// TIA Portal V20 export
DATA_BLOCK "Interface"   // DB238
{ S7_Optimized_Access := 'TRUE' }
// stored: MemoryReserve 0
   VAR
      enable : Bool;
      cont : Bool;
      localPort : UInt := 2000;
      interfaceId : HW_ANY := 120;
      connectionId : CONN_OUC := 16#1;
      reset : Bool;
      datasTemp : Array[0..181] of Byte;
      epcTemp : Array[0..127] of Byte;
      error : Bool;
      done : Bool;
      connected : Bool;
      restart : Bool;
      lenEpcId : Byte;
      lenData : Byte;
      status : Word;
      statusId : UInt;
      epcBuffer : Array[0..31, 0..127] of Byte;
      dataBuffer : Array[0..31, 0..181] of Byte;
      bufferIndex : Int;
      fillPattern : Byte;
   END_VAR
BEGIN
END_DATA_BLOCK
